# EPICS autosave request: iocBoot/ioc13Linux/auto_positions.req
file "CARS_motor_positions.req",         P=13Linux:, M=m1
file "CARS_motor_positions.req",         P=13Linux:, M=m2
file "CARS_motor_positions.req",         P=13Linux:, M=m3
~
